FUNCTION_BLOCK FB_FileWriter // Helper function block that writes to CSV files. 
VAR_INPUT
	sFilePath	: T_MaxString; 
	sFileName	: T_MaxString; 
	sNetID		: STRING; // NetID of the target, leave empty for local
END_VAR
VAR
	fbFileOpen : FB_FileOpen; 
	fbFilePuts : FB_FilePuts; 
	fbFileClose : FB_FileClose; 
	nFileHandle : UINT; 
	
	arrBuffer : ARRAY[0..100] OF T_MaxString; 
	eFileWriteState : (IDLE, OPEN_FILE, WRITE_TO_FILE, CLOSE_FILE, ERROR); 
END_VAR

CASE eFileWriteState OF
	IDLE: 
		// Make sure all the file writing FBs are ready for use (trigger on execute)
		Init(); 
		
		// We have pending data to be written 
		IF arrBuffer[0] <> '' THEN
			eFileWriteState := OPEN_FILE; 
		END_IF

	OPEN_FILE: 
	
		// Opens a file for writing at the end of the file (append). 
		// If the file does not exist, a new file is created. 
		fbFileOpen(
			bExecute		:= TRUE, 
			sNetID			:= sNetID, 
			sPathName		:= CONCAT(sFilePath, sFileName),
			nMode			:= FOPEN_MODEAPPEND); 
			
		IF fbFileOpen.bError THEN 
			eFileWriteState := ERROR; 
		ELSIF NOT fbFileOpen.bBusy THEN
			nFileHandle := fbFileOpen.hFile; 
			fbFileOpen(bExecute := FALSE); 
			eFileWriteState := WRITE_TO_FILE; 
		END_IF
		
	WRITE_TO_FILE: 
		fbFilePuts(
			bExecute		:= TRUE, 
			sNetId			:= sNetId, 
			hFile 			:= nFileHandle,
			sLine			:= arrBuffer[0]);
		
		IF fbFilePuts.bError THEN 
			eFileWriteState := ERROR; 
		ELSIF NOT fbFileClose.bBusy THEN
			// Sucess, data was written 
			//Rotate the buffer and close the file
			RotateBuffer(); 
			eFileWriteState := CLOSE_FILE; 
		END_IF
		
	CLOSE_FILE: 
		fbFileClose(
			bExecute		:= TRUE, 
			sNetId			:= sNetId, 
			hFile			:= nFileHandle); 
			
		IF fbFileClose.bError THEN
			eFileWriteState := ERROR; 
		ELSIF NOT fbFileClose.bBusy THEN
			nFileHandle := 0; 
			eFileWriteState := IDLE; 
		END_IF
		
	ERROR: 
		// Error, clear the handle and go back to idle 
		nFileHandle := 0;
		eFileWriteState := IDLE; 
END_CASE

METHOD PRIVATE Init : BOOL
VAR_INPUT
END_VAR
fbFileClose(bExecute := FALSE); 
fbFileOpen(bExecute := FALSE); 
fbFilePuts(bExecute := FALSE);
END_METHOD

METHOD PRIVATE InsertToBuffer
VAR_INPUT
	value	: STRING;
END_VAR
VAR
	nBufferIndex	: INT; 
END_VAR
FOR nBufferIndex := 0 TO 100 BY 1 DO
	IF arrBuffer[nBufferIndex] = '' THEN 
		// We foudn the free spot in the buffer, insert the value to this place 
		arrBuffer[nBufferIndex] := value;
		EXIT;
	END_IF
END_FOR
END_METHOD

METHOD PRIVATE RotateBuffer
VAR
	nIndex	: INT := 0; 
END_VAR
FOR nIndex := 0 TO 99 BY 1 DO
	// We can exit when we reached the empty slot in the buffer 
	IF arrBuffer[nIndex] = '' THEN
		EXIT; 
	END_IF
	// FIFO, removing first element in the array copying the next, etc...
	arrBuffer[nIndex] := arrbuffer[nIndex + 1]; 
END_FOR
END_METHOD

METHOD WriteToFile : BOOL
VAR_INPUT
	message : T_MaxString; 
END_VAR
InsertToBuffer(value := message);
END_METHOD

END_FUNCTION_BLOCK

(* stored: Version 1.1.0.1, ProductVersion 3.1.4024.12
   POU FB_FileWriter: Id {0e3b578c-6bd4-4984-b82b-3afa418d92c0}, SpecialFunc None
   Method Init: Id {471f8322-2af0-4ad6-9cd9-466774d1dcf5}
   Method InsertToBuffer: Id {6c567c6f-ce74-4640-8ccc-7ca4c5b1ccaf}
   Method RotateBuffer: Id {1d1ebc99-7968-499c-ba41-c54703d37556}
   Method WriteToFile: Id {555c72a9-c2ed-4ca8-8b20-a4d2fb75f41e} *)
